ABB RobotStudio station: mySolution2_20200830-185713.rsstn

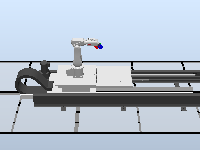
Station mySolution2 (saved by RobotStudio 20.1.9014.1)
Controller Controller1
  mechanical unit ROB_1: IRB120_3_58__01, 6 joints, base frame (0, 0, 397.5) mm
  mechanical unit TRACK: RTT_Bobin_1_7, 1 joints, base frame (0, 0, 397.5) mm
Layout (positions relative to the parent item):
  - RTT_Bobin_1_7 [mechanism] at (0, 0, 0) mm; joint values [0] (rad or m)
      links: Base, Link1
  - IRB120_3_58__01 [mechanism, from Robots\IRB120_3_58_G_01.rslib] at (0, 0, 397.5) mm; joint values [0, 0, 0, 0, 0.8098, 0] (rad or m)
Attachment: IRB120_3_58__01 is attached to RTT_Bobin_1_7 / Link1
